FUNCTION_BLOCK L2_Evacuador_SFC EXTENDS L1_ControllerBase_SFC

VAR_INPUT 				// Sensores y comandos
	Evacuar		: BOOL; // Hay que evacuar la tapa en la posición del módulo
	f0        	: BOOL; (* gh0 (nombre=f0  c=I22 B=J2 b=22 módulo=EL1008 T=6  C=6 etiqueta=-B10, input) Pick and place de rechazo detrás *)
    f1        	: BOOL; (* gh1 (nombre=f1  c=I23 B=J2 b=06 módulo=EL1008 T=6  C=6 etiqueta=-B11, input) Pick and place de rechazo delante *)
    g0        	: BOOL; (* gv1 (nombre=g0  c=I24 B=J2 b=31 módulo=EL1008 T=6  C=6 etiqueta=-B12, input) Pick and place de rechazo arriba *)
    v1        	: BOOL; (* ge1 (nombre=v1  c=I25 B=J1 b=25 módulo=EL1008 T=7  C=7 etiqueta=-B13, input) Pick and place de rechazo vacío *)
END_VAR

VAR_OUTPUT				// Actuadores
	F_1       	: BOOL; (* gHRA (nombre=F+  c=Q22 B=J2  b=35 módulo=EL2008 T=8 C=8 etiqueta=-Y8,  output) Pick and place de rechazo avanza (afuera) *)
    F_0       	: BOOL; (* gHRR (nombre=F-  c=Q23 B=J2  b=32 módulo=EL2008 T=8 C=8 etiqueta=-Y9,  output) Pick and place de rechazo retrocede *)
    G_1       	: BOOL; (* gVER (nombre=G+  c=Q24 B=J2  b=11 módulo=EL2008 T=8 C=8 etiqueta=-Y10, output) Pick and place de rechazo baja *)
    V_1       	: BOOL; (* gEYE (nombre=V+  c=Q25 B=J2  b=08 módulo=EL2008 T=9 C=9 etiqueta=-Y11, output) Pick and place de rechazo succiona *)
END_VAR

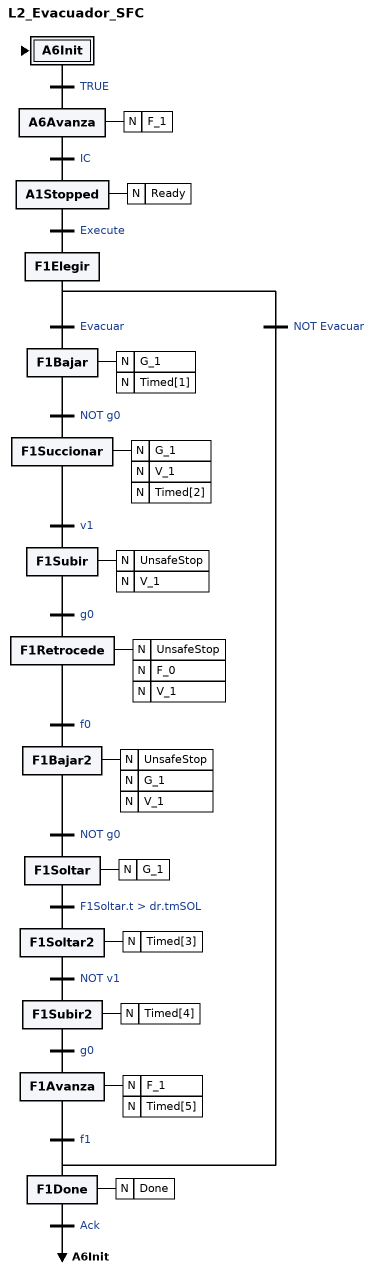
INITIAL_STEP A6Init:
END_STEP
TRANSITION FROM A6Init TO A6Avanza
    := TRUE;
END_TRANSITION
STEP A6Avanza:
    F_1(N);
END_STEP
TRANSITION FROM A6Avanza TO A1Stopped
    := IC;
END_TRANSITION
STEP A1Stopped:
    Ready(N);
END_STEP
TRANSITION FROM A1Stopped TO F1Elegir
    := Execute;
END_TRANSITION
STEP F1Elegir:
END_STEP
TRANSITION FROM F1Elegir TO F1Bajar
    := Evacuar;
END_TRANSITION
STEP F1Bajar:
    G_1(N);
    Timed[1](N);
END_STEP
TRANSITION FROM F1Bajar TO F1Succionar
    := NOT g0;
END_TRANSITION
STEP F1Succionar:
    G_1(N);
    V_1(N);
    Timed[2](N);
END_STEP
TRANSITION FROM F1Succionar TO F1Subir
    := v1;
END_TRANSITION
STEP F1Subir:
    UnsafeStop(N);
    V_1(N);
END_STEP
TRANSITION FROM F1Subir TO F1Retrocede
    := g0;
END_TRANSITION
STEP F1Retrocede:
    UnsafeStop(N);
    F_0(N);
    V_1(N);
END_STEP
TRANSITION FROM F1Retrocede TO F1Bajar2
    := f0;
END_TRANSITION
STEP F1Bajar2:
    UnsafeStop(N);
    G_1(N);
    V_1(N);
END_STEP
TRANSITION FROM F1Bajar2 TO F1Soltar
    := NOT g0;
END_TRANSITION
STEP F1Soltar:
    G_1(N);
END_STEP
TRANSITION FROM F1Soltar TO F1Soltar2
    := F1Soltar.t > dr.tmSOL;
END_TRANSITION
STEP F1Soltar2:
    Timed[3](N);
END_STEP
TRANSITION FROM F1Soltar2 TO F1Subir2
    := NOT v1;
END_TRANSITION
STEP F1Subir2:
    Timed[4](N);
END_STEP
TRANSITION FROM F1Subir2 TO F1Avanza
    := g0;
END_TRANSITION
STEP F1Avanza:
    F_1(N);
    Timed[5](N);
END_STEP
TRANSITION FROM F1Avanza TO F1Done
    := f1;
END_TRANSITION
TRANSITION FROM F1Elegir TO F1Done
    := NOT Evacuar;
END_TRANSITION
STEP F1Done:
    Done(N);
END_STEP
TRANSITION FROM F1Done TO A6Init
    := Ack;
END_TRANSITION

END_FUNCTION_BLOCK

(* stored: Version 1.1.0.1, ProductVersion 3.1.4024.11
   POU L2_Evacuador_SFC: Id {732a5d89-d610-4122-b553-0a1448cdc8d0}, SpecialFunc None *)
